// TIA Portal V21 export
VAR_GLOBAL   // PLC tag table "InputDigitali"
   CentralinaEmergenzeOk AT %I0.0 : Bool;   // Steuergerätnotfälleok / Control unitemergenzeok / Centralitaemergenciasok / Unité d'urgenceok / Centralinaemergenzeok
   PulsanteEmergenzaQE AT %I0.1 : Bool;   // Not-aus-tasteqe / Qeeeemergencybutton / Botónemergenciaqe / Bouton d'urgenceqe / Pulsanteemergenzaqe
   PulsanteEmergenzaRemoto AT %I0.2 : Bool;   // Not-ausrückstelltaste / Remoteemergencybutton / Botónemergenciaremoto / Bouton d'urgenceremoto / Pulsanteemergenzaremoto
   "E0.3" AT %I0.3 : Bool;   // E0.3
   TeleruttoreGenerale AT %I0.4 : Bool;
   "E0.5" AT %I0.5 : Bool;
   PressostatoBarilottoAcquaCalda AT %I0.6 : Bool;
   PressostatoAria AT %I0.7 : Bool;
   PulsanteMarciaCiclo AT %I1.0 : Bool;
   PulsanteComandoRecupero AT %I1.1 : Bool;
   PulsanteReset AT %I1.2 : Bool;
   PulsanteStopCiclo AT %I1.3 : Bool;
   LivelloSerbatoioCaldo_Max AT %I1.4 : Bool;
   LivelloSerbatoioCaldo_Min AT %I1.5 : Bool;
   PompaOlio_PressostatoMinima AT %I1.6 : Bool;
   PompaOlio_PressostatoMassima AT %I1.7 : Bool;
   Agitatore_TermicoOk AT %I2.0 : Bool;
   PompaMono_Ready AT %I2.1 : Bool;
   PompaMono_Servoventola_TermicoOk AT %I2.2 : Bool;
   CentrifugaLavaggio_TermicoOk AT %I2.3 : Bool;
   PompaPistoni_Ready AT %I2.4 : Bool;
   PompaPistoni_Ventola_TermicoOk AT %I2.5 : Bool;
   PompaOlio_TermicoOk AT %I2.6 : Bool;
   PompaRicircoloAcqua_TermicoOk AT %I2.7 : Bool;
   PompaRilancioTorre_Ready AT %I3.0 : Bool;
   PompaPistoni_Aspiratore_TermicoOk AT %I3.1 : Bool;
   "E3.2" AT %I3.2 : Bool;
   "E3.3" AT %I3.3 : Bool;
   "E3.4" AT %I3.4 : Bool;
   ValvolaB_SensoreAperto AT %I3.5 : Bool;   // Produzione
   ValvolaB_SensoreChiuso AT %I3.6 : Bool;   // Riciclo
   Flowmeter_ImpulsoTotalizzatore AT %I3.7 : Bool;
   Agitatore_Marcia AT %I4.0 : Bool;
   PompaMono_Marcia AT %I4.1 : Bool;
   CentrifugaLavaggio_Marcia AT %I4.2 : Bool;
   PompaPistoni_Marcia AT %I4.3 : Bool;
   PompaOlio_Marcia AT %I4.4 : Bool;
   PompaRicircoloAcqua_Marcia AT %I4.5 : Bool;
   PompaRilancioTorre_Marcia AT %I4.6 : Bool;
   "E4.7" AT %I4.7 : Bool;
   Consenso_DaCFT_SterilizzazioneTerminata AT %I5.0 : Bool;
   Consenso_DaCFT_SterilizzazioneInCorso AT %I5.1 : Bool;
   Consenso_DaCFT_LavaggioInCorso AT %I5.2 : Bool;
   Consenso_DaCFT_DosaggioInCorso AT %I5.3 : Bool;
   Consenso_DaCFT_RiempitriceInProduzione AT %I5.4 : Bool;
   Consenso_DaCFT_TemperaturaSterilizzazioneOk AT %I5.5 : Bool;
   "E5.6" AT %I5.6 : Bool;
   "E5.7" AT %I5.7 : Bool;
END_VAR
